{attribute 'qualified_only'}
{attribute 'strict'}
TYPE E_WinchMode :
(
	SETTLED := 0,
	ENGAGED
) USINT;
END_TYPE

(* stored: Version 1.1.0.1, ProductVersion 3.1.4022.18
   DUT E_WinchMode: Id {89b45946-b5a0-47d6-ab29-c727b3e6de70} *)
